(* IEC 61131-3 sources: template-ax2tia/template/src, 4 files *)

(* ---- myFunction.st ---- *)
NAMESPACE Simatic.Ax.DemoLibrary
    FUNCTION myFunction
        ;
    END_FUNCTION;
END_NAMESPACE

(* ---- Example.st ---- *)
NAMESPACE Simatic.Ax.DemoLibrary
    CLASS ExampleClass
        VAR PUBLIC

        END_VAR
        VAR PROTECTED
            _value : DINT;
        END_VAR

        METHOD PUBLIC RunCyclic
            _value := _value + DINT#1;
        END_METHOD

        METHOD PUBLIC GetValue : DINT
            GetValue := _value;
        END_METHOD

    END_CLASS
END_NAMESPACE

(* ---- myClass.st ---- *)
NAMESPACE Simatic.Ax.DemoLibrary
    CLASS myClass
        VAR

        END_VAR

    END_CLASS

END_NAMESPACE

(* ---- WrapperFB.st ---- *)
NAMESPACE Simatic.Ax.DemoLibrary
    FUNCTION_BLOCK WrapperFB
        VAR_INPUT
            Enable : BOOL;
        END_VAR
        VAR_OUTPUT
            Counts : DINT;
        END_VAR
        VAR
           _inst : ExampleClass;
           _cyclesCounted : INT;
        END_VAR

        _inst.RunCyclic();
        Counts := _inst.GetValue();
    END_FUNCTION_BLOCK
END_NAMESPACE
